// TIA Portal V19 export
DATA_BLOCK "A0302_HU_Cytropack_PERS"   // DB195
// stored: MemoryReserve 100
   VAR RETAIN
      Par : Struct
         Bloccaggio : Struct
            TargetPressure : Real := 100.0;
            TargetMaxSpeed : Real := 3000.0;
            Delta : Struct
               Min : Real := 0.5;
               Max : Real := 0.5;
            END_STRUCT;
         END_STRUCT;
         Pareggiamento : Struct
            TargetPressure : Real := 100.0;
            TargetMaxSpeed : Real := 3000.0;
            Delta : Struct
               Min : Real := 0.5;
               Max : Real := 0.5;
            END_STRUCT;
         END_STRUCT;
      END_STRUCT;
   END_VAR
BEGIN
END_DATA_BLOCK
